TYPE Machine :
STRUCT
	
	carriageIsUp : BOOL := FALSE; (* Carriage is in the "up" position *)
	carriageIsDown : BOOL := FALSE; (* Carriage is in the "down" position *)
	zero : BOOL := FALSE; (* Machine has been zero'd *)
		
END_STRUCT
END_TYPE

(* stored: Version 1.1.0.1, ProductVersion 3.1.4024.3
   DUT Machine: Id {a16ac569-0aaa-4e8a-811f-9e420ea2f988} *)
